{attribute 'enable_dynamic_creation'}
FUNCTION_BLOCK FB_Robot6Axis EXTENDS FB_Robot
VAR
	// 6 Axis Robot Properties
	currentTool : STRING(80); // TODO: Replace with TOOL type when defined
	currentFrame : STRING(80); // TODO: Replace with FRAME type when defined
	currentFrameId : INT;
	jointPosition : ST_JointPosition6;
	jointVelocity : ST_JointPosition6;
	TCPPosition : ST_Pose3D;
	TCPVelocity : ST_Pose3D;
	isInHomePosition : BOOL;
	isInCollision : BOOL;
	// Cam: Camera // TODO: Add camera reference
END_VAR

// 6 Axis Robot implementation

METHOD PUBLIC Home : BOOL
VAR_INPUT
END_VAR
// Move robot to home position
END_METHOD

METHOD PUBLIC SwitchTool : BOOL
VAR_INPUT
	tool : STRING(80); // TODO: Replace with TOOL type when defined
END_VAR
currentTool := tool;
END_METHOD

END_FUNCTION_BLOCK

(* stored: Version 1.1.0.1
   POU FB_Robot6Axis: Id {f1b2c3d4-2222-2222-2222-222222222222}
   Method Home: Id {f1b2c3d4-2221-2222-2222-222222222222}
   Method SwitchTool: Id {f1b2c3d4-2222-2222-2222-222222222222} *)
